FUNCTION_BLOCK Puls

VAR_INPUT
 	EN 		:BOOL := TRUE;
    Period	:TIME;
END_VAR
VAR_OUTPUT
	Puls	:BOOL;
END_VAR
VAR
	M		:BOOL:=0;
	R1		:R_TRIG;
	t		:BOOL;
	R2		:R_TRIG;
	TP1		:TP;
	TP2		:TP;
	M1		:BOOL:=0;
END_VAR

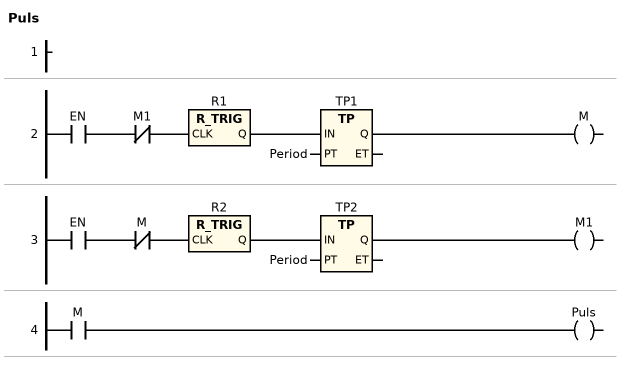
// NETWORK 1

// NETWORK 2
R1(CLK := EN AND NOT M1); // R_TRIG
TP1(IN := R1.Q, PT := Period); // TP
M := TP1.Q;

// NETWORK 3
R2(CLK := EN AND NOT M); // R_TRIG
TP2(IN := R2.Q, PT := Period); // TP
M1 := TP2.Q;

// NETWORK 4
Puls := M;

END_FUNCTION_BLOCK

(* stored: Version 1.1.0.1, ProductVersion 3.1.4024.4
   POU Puls: Id {ae56ab5d-2644-4886-9eea-e4c2f88efcb1}, SpecialFunc None *)
